(* PLC project SafeLOGIC-1, BrAutomation SafeDESIGNER  4.4.0.0 *)
(* stored: companyURL http://www.br-automation.com, creationDateTime Tue Oct 19 12:10:16 2021 *)

PROGRAM Main
  VAR  (* added by the conversion: wires and edge detectors of the diagram *)
    _SAFEBOOL_TO_BOOL81_OUT : BOOL;
  END_VAR

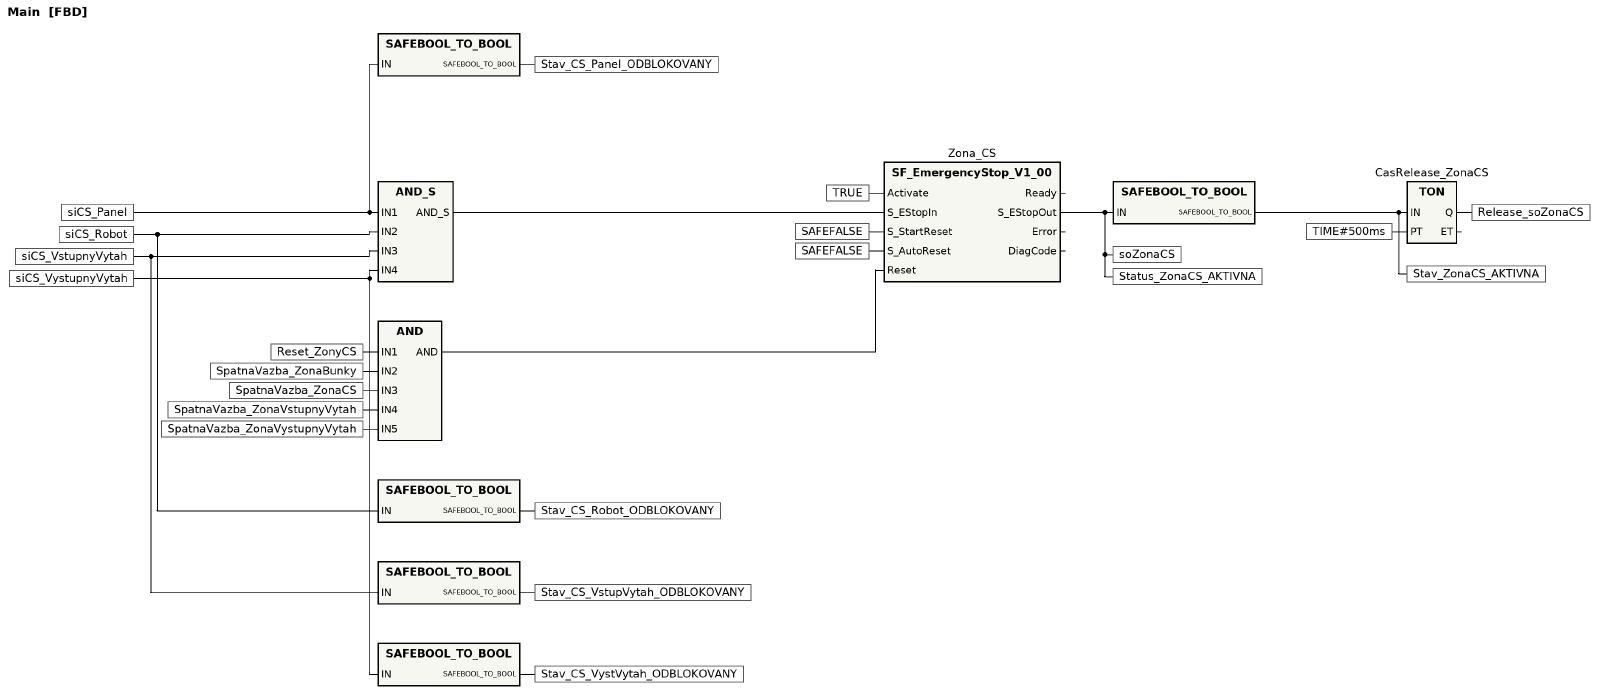
(* FBD diagram, written out as Structured Text *)
Stav_CS_Panel_ODBLOKOVANY := SAFEBOOL_TO_BOOL(siCS_Panel);
Zona_CS(Activate := TRUE, S_EStopIn := AND_S(siCS_Panel, siCS_Robot, siCS_VstupnyVytah, siCS_VystupnyVytah), S_StartReset := SAFEFALSE, S_AutoReset := SAFEFALSE, Reset := Reset_ZonyCS AND SpatnaVazba_ZonaBunky AND SpatnaVazba_ZonaCS AND SpatnaVazba_ZonaVstupnyVytah AND SpatnaVazba_ZonaVystupnyVytah);
soZonaCS := Zona_CS.S_EStopOut;
Status_ZonaCS_AKTIVNA := Zona_CS.S_EStopOut;
Stav_CS_Robot_ODBLOKOVANY := SAFEBOOL_TO_BOOL(siCS_Robot);
_SAFEBOOL_TO_BOOL81_OUT := SAFEBOOL_TO_BOOL(Zona_CS.S_EStopOut);
CasRelease_ZonaCS(IN := _SAFEBOOL_TO_BOOL81_OUT, PT := TIME#500ms);
Release_soZonaCS := CasRelease_ZonaCS.Q;
Stav_CS_VstupVytah_ODBLOKOVANY := SAFEBOOL_TO_BOOL(siCS_VstupnyVytah);
Stav_ZonaCS_AKTIVNA := _SAFEBOOL_TO_BOOL81_OUT;
Stav_CS_VystVytah_ODBLOKOVANY := SAFEBOOL_TO_BOOL(siCS_VystupnyVytah);
END_PROGRAM
